Staubli VAL3: getMoveType.pgx

public program getMoveType(num& x_nMoveType[], num x_nIndex, bool x_bCycle)
begin
  // get the moveType
  if x_bCycle
    x_nMoveType=pt:tTraj[sTrajCycle].tData[x_nIndex].tSuper.moveType
  else
    x_nMoveType=jEditPoint.tData[x_nIndex].tSuper.moveType
  endIf
end
